// TIA Portal V17 export
// export: Created 2024-06-25T12:57:18.3598068Z, ExportSetting WithDefaults, DisplayName Totally Integrated Automation Portal, DisplayVersion V17 Update 6, DisplayName TIA Portal Openness, DisplayVersion V17 Update 6, DisplayName TIA Portal Version Control Interface, DisplayVersion V17, DisplayName STEP 7 Professional, DisplayVersion V17 Update 6, DisplayName STEP 7 Safety, DisplayVersion V17 Update 6, DisplayName WinCC Advanced, DisplayVersion V17 Update 6
FUNCTION "Res" : Void   // FC1, LAD
{ S7_Optimized_Access := 'TRUE' }
VERSION : 0.1
// stored: AutoNumber true, IsIECCheckEnabled false, SetENOAutomatically false, UDAEnableTagReadback false
BEGIN

REGION Network 1: PULSADOR OFF
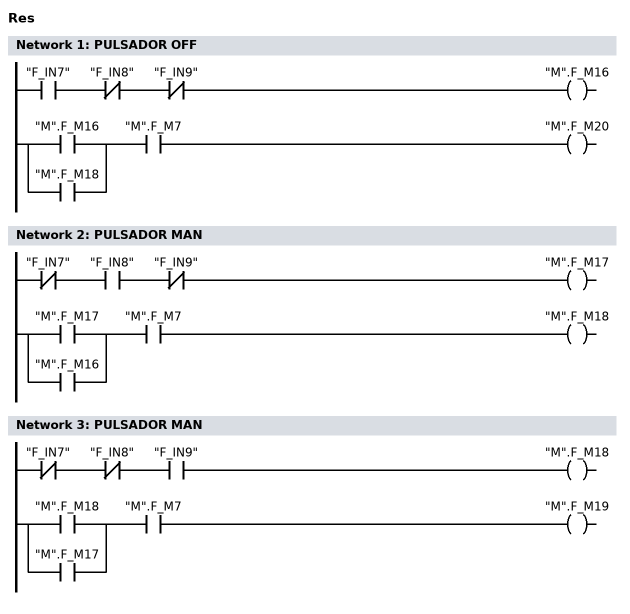
   RUNG wire#powerrail
      Contact( "F_IN7" )
      I_Contact( "F_IN8" )
      I_Contact( "F_IN9" )
      Coil( "M".F_M16 )
   END_RUNG
   RUNG wire#powerrail
      Contact( "M".F_M16 )
      wire#w1
      Contact( "M".F_M7 )
      Coil( "M".F_M20 )
   END_RUNG
   RUNG wire#powerrail
      Contact( "M".F_M18 )
   END_RUNG wire#w1
   // the same network as SCL:
   "M".F_M16 := "F_IN7" AND NOT "F_IN8" AND NOT "F_IN9";
   "M".F_M20 := ("M".F_M16 OR "M".F_M18) AND "M".F_M7;
END_REGION

REGION Network 2: PULSADOR MAN
   RUNG wire#powerrail
      I_Contact( "F_IN7" )
      Contact( "F_IN8" )
      I_Contact( "F_IN9" )
      Coil( "M".F_M17 )
   END_RUNG
   RUNG wire#powerrail
      Contact( "M".F_M17 )
      wire#w1
      Contact( "M".F_M7 )
      Coil( "M".F_M18 )
   END_RUNG
   RUNG wire#powerrail
      Contact( "M".F_M16 )
   END_RUNG wire#w1
   // the same network as SCL:
   "M".F_M17 := NOT "F_IN7" AND "F_IN8" AND NOT "F_IN9";
   "M".F_M18 := ("M".F_M17 OR "M".F_M16) AND "M".F_M7;
END_REGION

REGION Network 3: PULSADOR MAN
   RUNG wire#powerrail
      I_Contact( "F_IN7" )
      I_Contact( "F_IN8" )
      Contact( "F_IN9" )
      Coil( "M".F_M18 )
   END_RUNG
   RUNG wire#powerrail
      Contact( "M".F_M18 )
      wire#w1
      Contact( "M".F_M7 )
      Coil( "M".F_M19 )
   END_RUNG
   RUNG wire#powerrail
      Contact( "M".F_M17 )
   END_RUNG wire#w1
   // the same network as SCL:
   "M".F_M18 := NOT "F_IN7" AND NOT "F_IN8" AND "F_IN9";
   "M".F_M19 := ("M".F_M18 OR "M".F_M17) AND "M".F_M7;
END_REGION
END_FUNCTION
